{attribute 'pack_mode' := '1'}
TYPE ST_OutputArgInfoAndData :
STRUCT
	nNumberOfOutputArguments: UDINT; // determined amount of output parameters
	nReserved: ARRAY[1..4] OF BYTE; // Reserved padding
	stOutputArgInfo: ARRAY[1..2] OF ST_UAMethodArgInfo; // number of output parameters - this method has 2 output parameter 
	out1: INT;
	out2 : DINT;
END_STRUCT
END_TYPE

(* stored: Version 1.1.0.1
   DUT ST_OutputArgInfoAndData: Id {aa411b33-0ffd-48f8-ad37-0dd63243bc1d} *)
